PROGRAM BackgroundCOM
VAR
	i : DINT;
	

END_VAR

FOR i := 0 TO 2 DO
	IMU.fbStim300[i](fJointAccAtImuX := MAIN.fGainAccXYZ[0]*MAIN.AccelerometerReadingsOutWithoutGravity[i].X/CONSTANTS.GRAVITY,//represent in terms of Gravuty constant
					fJointAccAtImuY := MAIN.fGainAccXYZ[1]*MAIN.AccelerometerReadingsOutWithoutGravity[i].Y/CONSTANTS.GRAVITY,
					fJointAccAtImuZ := MAIN.fGainAccXYZ[2]*MAIN.AccelerometerReadingsOutWithoutGravity[i].Z/CONSTANTS.GRAVITY);
END_FOR

END_PROGRAM

(* stored: Version 1.1.0.1, ProductVersion 3.1.4024.9
   POU BackgroundCOM: Id {b271819f-2bcd-49a4-b99d-11668f790144}, SpecialFunc None *)
